FUNCTION TryConvert_WORD_TO_UINT : BOOL
VAR_INPUT
	in : WORD;
	out : REFERENCE TO UINT;
END_VAR

out := WORD_TO_UINT(in);
TryConvert_WORD_TO_UINT := TRUE;

END_FUNCTION

(* stored: Version 1.1.0.1, ProductVersion 3.1.4024.12
   POU TryConvert_WORD_TO_UINT: Id {87d5fd9e-6055-4e7f-a103-e24a731195b3}, SpecialFunc None *)
